FUNCTION_BLOCK TabletFillingControl02
VAR_INPUT
	MachineStart				:	BOOL;		// True=Machine On
	FillingPosition				:	BOOL;		// Tube in loading position
	TabletsInTube				:	UINT;		// Number of tablets which should be loaded into one tube
	LightBarrier				:	BOOL;		// False=free (no tablet present), True=tablet present
END_VAR
VAR_OUTPUT
	BeltMotorCmdOn				:	BOOL;		// Belt motor command ON
	ValveCmdOpen				:	BOOL;		// Valve command OPEN
	TabletsSelected				:	UINT;		// Number of tablet selected to be loaded into one tube
END_VAR
VAR
	ctdTablets					: CTD;		// down counter for three tablets
	
	FirstScan					: BOOL;
	OneShot						: BOOL;		// one shot pulse after power restart		
	srTabletNumberSelected		: SR;		// Number of tablets properly selected (>0)

	WAIT						: BOOL;		// Machine state 'Wait'
	SWITCHED_ON					: BOOL;		// Machine state 'Switched on'
	WAIT_FOR_FILL_POS			: BOOL;		// Machine state 'Waiting for filling position'
	FILL_POS_REACHED			: BOOL;		// Machine state 'Filling position reached'
	LOAD_CTR_TABLETS			: BOOL;		// Machine state 'Load counter with tablets number'

	
	rtTabletCntrLoaded			: R_TRIG;	// Tablet counter loaded with number of tablet
	tonCountTablet				: TON;		// delay after last tablet detected to allow proper positioning in the tube
END_VAR
VAR // added by the converter: edge detectors and wires of the graphical bodies
    _w1 : BOOL;
END_VAR

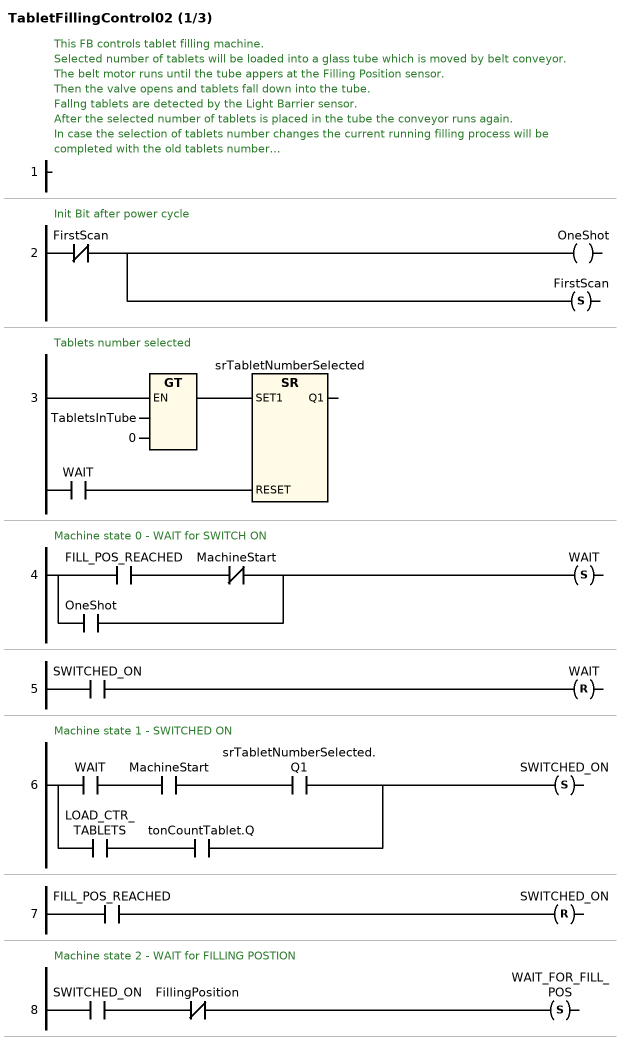
// NETWORK 1
// This FB controls tablet filling machine.
// Selected number of tablets will be loaded into a glass tube which is moved by belt conveyor.
// The belt motor runs until the tube appers at the Filling Position sensor.
// Then the valve opens and tablets fall down into the tube.
// Fallng tablets are detected by the Light Barrier sensor.
// After the selected number of tablets is placed in the tube the conveyor runs again.
// In case the selection of tablets number changes the current running filling process will be completed with the old tablets number.
// This is Version 02 of the program - any number number of tablets can be chosen by 'TabletsInTube' variable

// NETWORK 2
// Init Bit after power cycle
_w1 := NOT FirstScan;
OneShot := _w1;
FirstScan S= _w1;

// NETWORK 3
// Tablets number selected
srTabletNumberSelected(SET1 := TabletsInTube > 0, RESET := WAIT); // SR

// NETWORK 4
// Machine state 0 - WAIT for SWITCH ON
WAIT S= FILL_POS_REACHED AND NOT MachineStart OR OneShot;

// NETWORK 5
WAIT R= SWITCHED_ON;

// NETWORK 6
// Machine state 1 - SWITCHED ON
SWITCHED_ON S= WAIT AND MachineStart AND srTabletNumberSelected.Q1 OR LOAD_CTR_TABLETS AND tonCountTablet.Q;

// NETWORK 7
SWITCHED_ON R= FILL_POS_REACHED;

// NETWORK 8
// Machine state 2 - WAIT for FILLING POSTION
WAIT_FOR_FILL_POS S= SWITCHED_ON AND NOT FillingPosition;

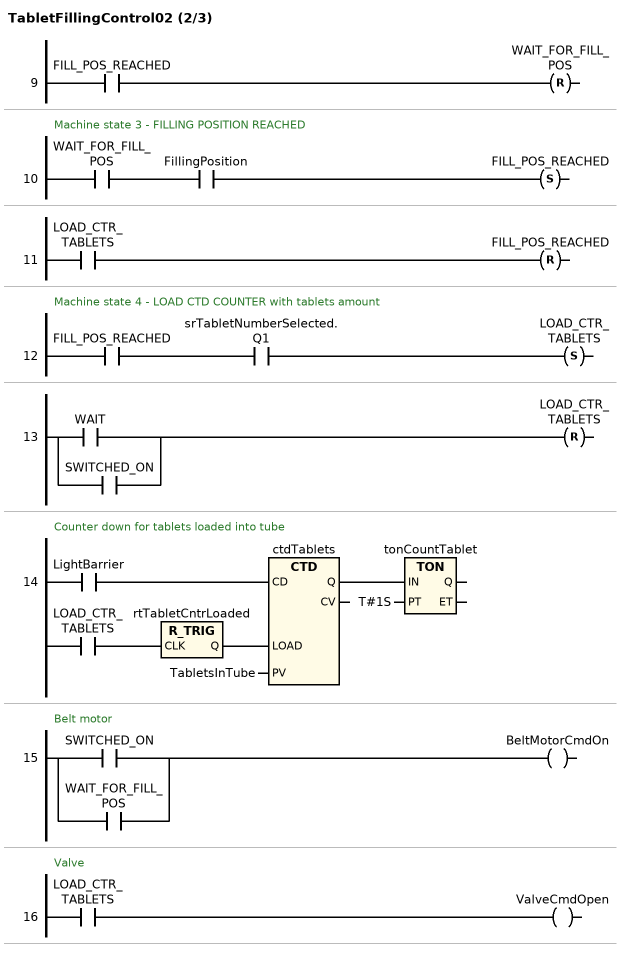
// NETWORK 9
WAIT_FOR_FILL_POS R= FILL_POS_REACHED;

// NETWORK 10
// Machine state 3 - FILLING POSITION REACHED
FILL_POS_REACHED S= WAIT_FOR_FILL_POS AND FillingPosition;

// NETWORK 11
FILL_POS_REACHED R= LOAD_CTR_TABLETS;

// NETWORK 12
// Machine state 4 - LOAD CTD COUNTER with tablets amount
LOAD_CTR_TABLETS S= FILL_POS_REACHED AND srTabletNumberSelected.Q1;

// NETWORK 13
LOAD_CTR_TABLETS R= WAIT OR SWITCHED_ON;

// NETWORK 14
// Counter down for tablets loaded into tube
rtTabletCntrLoaded(CLK := LOAD_CTR_TABLETS); // R_TRIG
ctdTablets(CD := LightBarrier, LOAD := rtTabletCntrLoaded.Q, PV := TabletsInTube); // CTD
tonCountTablet(IN := ctdTablets.Q, PT := T#1S); // TON

// NETWORK 15
// Belt motor
BeltMotorCmdOn := SWITCHED_ON OR WAIT_FOR_FILL_POS;

// NETWORK 16
// Valve
ValveCmdOpen := LOAD_CTR_TABLETS;

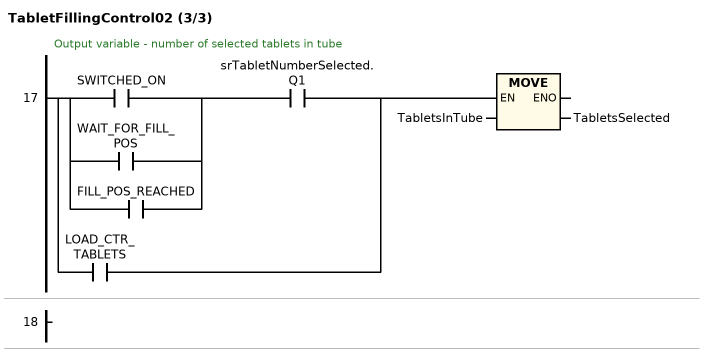
// NETWORK 17
// Output variable - number of selected tablets in tube
IF (SWITCHED_ON OR WAIT_FOR_FILL_POS OR FILL_POS_REACHED) AND srTabletNumberSelected.Q1 OR LOAD_CTR_TABLETS THEN
    TabletsSelected := TabletsInTube;
END_IF

// NETWORK 18

END_FUNCTION_BLOCK

(* stored: Version 1.1.0.1, ProductVersion 3.1.4024.15
   POU TabletFillingControl02: Id {e6d988ed-ae45-4ddc-9a89-612e781adffa}, SpecialFunc None *)
